SUBAPPLICATION Uebung_010d (* Toggle Flip-Flop mit IE SoftKey_F1 SK_RELEASED mit GreenWhiteBackground *)
  (* Standard: 61499-2; Description: Copyright (c) 2026 Meisterschulen am Ostbahnhof This program and the accompanying materials are made available under the terms of the Eclipse Public License 2.0 which is available at https://www.eclipse.org/legal/epl-2.0/ SPDX-License-Identifier: EPL-2.0 *)
  (* Version 1.0, 2026-09-02, Franz Höpfinger, Meisterschulen am Ostbahnhof, initial API and implementation and/or initial documentation *)
  PACKAGE Uebungen;
  IMPORT isobus::UT::io::Softkey::SoftKeyActivationCode::SK_RELEASED;
  IMPORT Uebungen::const::UT::DefaultPool::SoftKey_F1;
  IMPORT logiBUS::io::DQ::logiBUS_DO::Output_Q1;
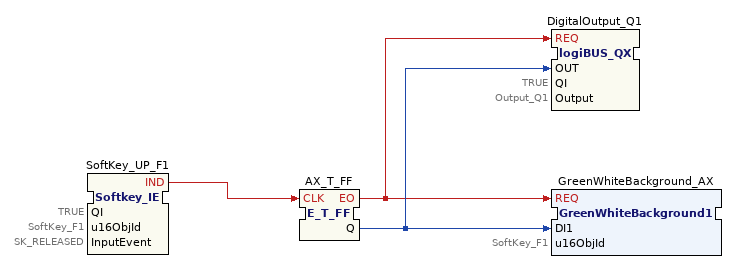
  FBS
    DigitalOutput_Q1 : logiBUS::io::DQ::logiBUS_QX(QI := TRUE, Output := Output_Q1);
    SoftKey_UP_F1 : isobus::UT::io::Softkey::Softkey_IE(QI := TRUE, u16ObjId := SoftKey_F1, InputEvent := SK_RELEASED);
    AX_T_FF : iec61499::events::E_T_FF;
  END_FBS
  SUBAPPS
    GreenWhiteBackground_AX : MyLib::sys::GreenWhiteBackground1(u16ObjId := SoftKey_F1);
  END_SUBAPPS
  EVENT_CONNECTIONS
    SoftKey_UP_F1.IND TO AX_T_FF.CLK;
    AX_T_FF.EO TO DigitalOutput_Q1.REQ;
    AX_T_FF.EO TO GreenWhiteBackground_AX.REQ;
  END_CONNECTIONS
  DATA_CONNECTIONS
    AX_T_FF.Q TO DigitalOutput_Q1.OUT;
    AX_T_FF.Q TO GreenWhiteBackground_AX.DI1;
  END_CONNECTIONS
END_SUBAPPLICATION
